FUNCTION_BLOCK FB_StateInit IMPLEMENTS I_State
VAR
	_refMainStateMachine		: REFERENCE TO FB_MainStateMachine;
END_VAR

METHOD StartButtonPressed
END_METHOD

METHOD StopButtonPressed
END_METHOD

METHOD SafetyAcknowledged
VAR_INPUT
END_VAR
END_METHOD

METHOD ClearErrors
END_METHOD

METHOD SafetyTripped
VAR_INPUT
END_VAR
_refMainStateMachine.SetState(_refMainStateMachine.ipStateEStop);
END_METHOD

METHOD FB_init : BOOL
VAR_INPUT
	// if TRUE, the retain variables are initialized (warm start / cold start)
	bInitRetains			: BOOL;
	// if TRUE, the instance afterwards gets moved into the copy code (online
	// change)
	bInCopyCode				: BOOL;
	fbMainStateMachine		: REFERENCE TO FB_MainStateMachine;
END_VAR
_refMainStateMachine REF= fbMainStateMachine;
END_METHOD

METHOD GetDescription : STRING
GetDescription := 'Initialization';
END_METHOD

METHOD Execute
END_METHOD

END_FUNCTION_BLOCK

(* stored: Version 1.1.0.1, ProductVersion 3.1.4024.11
   POU FB_StateInit: Id {0279ef55-8749-43f2-9b6d-b33bab30ffff}, SpecialFunc None
   Method StartButtonPressed: Id {259cd519-0d3b-4132-81ec-9e6582ef725a}
   Method StopButtonPressed: Id {5bcbd9e0-34b1-49d0-92cf-ebd7b40f9183}
   Method SafetyAcknowledged: Id {66a6e82f-44b9-4ef6-af53-489f9dbfbee4}
   Method ClearErrors: Id {8e286c84-0347-4016-a21c-8f3a83832f09}
   Method SafetyTripped: Id {b4ab07ef-9a3c-4938-a5af-d618d54e9104}
   Method FB_init: Id {bba99187-f902-4bd8-8cac-07377dad3116}
   Method GetDescription: Id {c64389ca-42c0-40d6-8412-1fd9d83f0279}
   Method Execute: Id {ffd65fcd-7940-4aad-813f-b77fa379a0dc} *)
